(* IEC 61131-3 sources: plcc/packages/plc-wasm/test/fixtures, 3 files *)

(* ---- div_zero.st ---- *)
(* SPDX-License-Identifier: MPL-2.0 *)
(* %MW0 is the divisor: 0 faults (integer division by zero). *)
PROGRAM Ratio
VAR
    divisor AT %MW0 : INT;
    lamp    AT %QX0.0 : BOOL;
    q       AT %MW1 : INT;
    after   : INT;
END_VAR
lamp := TRUE;
q := 100 / divisor;
after := after + 1;
END_PROGRAM

(* ---- seal_in.st ---- *)
(* SPDX-License-Identifier: MPL-2.0 *)
(* Motor seal-in: start latches the motor, stop drops it. *)
PROGRAM SealIn
VAR
    start AT %IX0.0 : BOOL;
    stop  AT %IX0.1 : BOOL;
    motor AT %QX0.0 : BOOL;
    starts AT %MW0  : UINT;
    runs  : DINT;
    level : REAL := 1.5;
    wave  : REAL;
    last  : BOOL;
    name  : STRING[16] := 'seal';
END_VAR
motor := (start OR motor) AND NOT stop;
IF motor AND NOT last THEN
    starts := starts + 1;
    PRINT('motor on');
END_IF;
last := motor;
runs := runs + 1;
wave := SIN(level);
END_PROGRAM

(* ---- ton.st ---- *)
(* SPDX-License-Identifier: MPL-2.0 *)
(* TON on %IX0.0 with PT = 500 ms; Q on %QX0.0, ET mirrored to %MD0 in ms. *)
CONFIGURATION Sim
    RESOURCE Cpu ON Wasm
        TASK Fast (INTERVAL := T#10ms, PRIORITY := 1);
        TASK Slow (INTERVAL := T#100ms, PRIORITY := 2);
        PROGRAM Main WITH Fast : Delay;
        PROGRAM Count WITH Slow : Counter;
    END_RESOURCE
END_CONFIGURATION

PROGRAM Delay
VAR
    go    AT %IX0.0 : BOOL;
    done  AT %QX0.0 : BOOL;
    et_ms AT %MD0   : UDINT;
    t : TON;
END_VAR
t(IN := go, PT := T#500ms);
done := t.Q;
et_ms := TIME_TO_UDINT(t.ET);
END_PROGRAM

PROGRAM Counter
VAR
    n AT %MW4 : UINT;
END_VAR
n := n + 1;
END_PROGRAM
